(* IEC 61131-3 sources: CodesysTest/alpha/export/FBs/Components/DelayDwellFB/DelayDwellFB.pou/DwellSetting.prop, 1 file *)

(* ---- Set.pm.st ---- *)
(*#-#-#-#-#-#-#-#-#-#---Declaration---#-#-#-#-#-#-#-#-#-#-#-#-#*)

VAR
END_VAR
(*#-#-#-#-#-#-#-#-#-#---Implementation---#-#-#-#-#-#-#-#-#-#-#-#-#*)

_dwellTimeInMS := DwellSetting;
